VAR_GLOBAL
	XAxisLimitSwPos AT %I* :BOOL;
	XAxisLimitSwNeg AT %I* :BOOL;
END_VAR

(* stored: Version 1.1.0.1, ProductVersion 3.1.4024.2
   GVL GVL_Sensors: Id {06d2cfb4-faea-47f7-8719-fc045936fbbb} *)
